FUNCTION F_CheckRollerDoor : BOOL
VAR_INPUT
	CurrentPos 		: REAL;
	RequestedPos 	: REAL;
	Door 			: sRollerDoor;
END_VAR
VAR
	DoorPos : REAL := 100000;
END_VAR

IF (CurrentPos < DoorPos AND RequestedPos > DoorPos) OR (CurrentPos > DoorPos AND RequestedPos < DoorPos) THEN
	Door.AutoOpenRequest := 1;
	IF Door.StatusOpenedInput THEN
		F_CheckRollerDoor := 1;
	END_IF
	ELSE
	F_CheckRollerDoor := 1;	
END_IF

END_FUNCTION

(* stored: Version 1.1.0.1, ProductVersion 3.1.4024.12
   POU F_CheckRollerDoor: Id {d7eec0a7-838b-4787-a890-8069ae873d55}, SpecialFunc None *)
